//--
// <ObjectWithoutContextExampleDeclaration>
(*
		
			This is an example of self-confident object, that initiate its context by itself.	

*)
FUNCTION_BLOCK Woltz_Object EXTENDS TcoCore.TcoObject
VAR
	//Horse owned by Jack Woltz.
	//https://godfather.fandom.com/wiki/Khartoum
	_Khartoum	: Horse_Object(THIS^);
END_VAR
//---------------------------------------------------------------------------
// </ObjectWithoutContextExampleDeclaration>
//--

METHOD FB_init : BOOL
VAR_INPUT
	bInitRetains : BOOL; // if TRUE, the retain variables are initialized (warm start / cold start)
	bInCopyCode : BOOL;  // if TRUE, the instance afterwards gets moved into the copy code (online change)
	Parent : ITcoObject;
END_VAR
END_METHOD

END_FUNCTION_BLOCK

(* stored: Version 1.1.0.1, ProductVersion 3.1.4024.6
   POU Woltz_Object: Id {210d7878-f3a8-0d74-1c18-c55600d21082}, SpecialFunc None
   Method FB_init: Id {da33549e-080b-0906-3324-f3717f68b2b3} *)
